{attribute 'Tc2GvlVarNames'}
VAR_GLOBAL CONSTANT
	(* BWK_Zustand_Status *)
	E_BWK_Zustand_Status_Idle_Sperre				: SINT := 0;
	E_BWK_Zustand_Status_Betriebsbereit				: SINT := 1;
	E_BWK_Zustand_Status_Nachl						: SINT := 2;
	E_BWK_Zustand_Status_Vorl						: SINT := 3;
	E_BWK_Zustand_Status_Betrieb					: SINT := 4;
	E_BWK_Zustand_Status_Betrieb_Sperre				: SINT := 5;
	E_BWK_Zustand_Status_Stoerung					: SINT := 99;

	(* BWK_Zustand_Regelung_Modus *)
	E_BWK_Regelung_Modus_P							: SINT := 0;
	E_BWK_Regelung_Modus_T							: SINT := 1;

	(* System_BWK_Zustand_Status *)
	E_System_BWK_Zustand_Status_Idle_Sperre			: SINT := 0;
	E_System_BWK_Zustand_Status_Betriebsbereit		: SINT := 1;
	E_System_BWK_Zustand_Status_Nachl_Stellventil	: SINT := 2;
	E_System_BWK_Zustand_Status_Vorl_Stellventil	: SINT := 3;
	(*E_System_BWK_Zustand_Status_Nachl_Pumpe		: SINT := 4;*)
	(*E_System_BWK_Zustand_Status_Vorl_Pumpe		: SINT := 5;*)
	E_System_BWK_Zustand_Status_Nachl_BWK			: SINT := 6;
	E_System_BWK_Zustand_Status_Vorl_BWK			: SINT := 7;
	E_System_BWK_Zustand_Status_Betrieb				: SINT := 8;
	E_System_BWK_Zustand_Status_Betrieb_Sperre		: SINT := 9;
	E_System_BWK_Zustand_Status_Stoerung			: SINT := 99;
END_VAR

(* stored: Version 1.1.0.1, ProductVersion 3.1.4024.9
   GVL Con_BWK: Id {dcf7ca45-5f89-4c31-860b-3ba98e334c97} *)
